PROGRAM MAIN

VAR
	(*
bEnable: BOOL := FALSE;
bMove: BOOL := FALSE;
fAxis1VelocityPercent: LREAL := 0;	
axis1: AXIS_REF;
fbAxis1Power: MC_Power;
fbAxis1MoveVelocity: MC_MoveVelocity;
MCDirectionAxis1 : MC_Direction;
fAxis1ReferenceVelocity: LREAL := 100;
*)

fbGetCurTaskIdx  : GETCURTASKINDEX;
nCycleTime       : UDINT;
END_VAR

P_Inputs();
P_MachineControl();
P_AxisControl();
P_Outputs();
P_StablePlatform();

fbGetCurTaskIdx();
nCycleTime := _TaskInfo[fbGetCurTaskIdx.index].CycleTime;

(*

bEnable := G_Inputs.bJoystickLeftEnable;
bMove := G_Inputs.bJoystickLeftEnable;
fAxis1VelocityPercent := ABS(G_Sensors.fJoystickLeftNormalizedX)*100;
MCDirectionAxis1 := G_Sensors.MCDirectionAxis1;

axis1.ReadStatus();

fbAxis1Power(
Axis:= axis1,
Enable:= bEnable,
Enable_Positive:= bEnable,
Enable_Negative:= bEnable,
Override:= fAxis1VelocityPercent,
BufferMode:= ,
Options:= ,
Status=> ,
Busy=> ,
Active=> ,
Error=> ,
ErrorID=> );

fbAxis1MoveVelocity(
Axis:= axis1,
Execute:= bMove,
Velocity:= fAxis1ReferenceVelocity,
Acceleration:= ,
Deceleration:= ,
Jerk:= ,
Direction:= G_Sensors.MCDirectionAxis1,
BufferMode:= ,
Options:= ,
InVelocity=> ,
Busy=> ,
Active=> ,
CommandAborted=> ,
Error=> ,
ErrorID=> );

*)

END_PROGRAM

(* stored: Version 1.1.0.1, ProductVersion 3.1.4024.12
   POU MAIN: Id {540b8970-e57b-4c7b-a65e-22bf2965a9b1}, SpecialFunc None *)
